// TIA Portal V17 export
// export: Created 2023-06-23T18:33:35.104452Z, ExportSetting WithDefaults, DisplayName Totally Integrated Automation Portal, DisplayVersion V17, DisplayName TIA Portal Openness, DisplayVersion V17, DisplayName TIA Portal Version Control Interface, DisplayVersion V17, DisplayName STEP 7 Professional, DisplayVersion V17, DisplayName STEP 7 Safety, DisplayVersion V17, DisplayName WinCC Advanced / Unified PC, DisplayVersion V17
DATA_BLOCK "ext"   // DB1
{ S7_Optimized_Access := 'FALSE' }
VERSION : 0.1
// stored: AutoNumber true, DBAccessibleFromOPCUA true, IsOnlyStoredInLoadMemory false, IsWriteProtectedInAS false
   VAR
      block : Bool := true;
      trig : USInt;
      switch : Array[1..17] of Bool;
      inv : Array[1..9] of Bool;
      aer : Array[1..8] of Bool;
      status : Array[1..32] of USInt;
   END_VAR
BEGIN
END_DATA_BLOCK
